(* LS Electric XG5000 project: Forward_Reverse *)
(* PLC LSPLC *)

PROGRAM NewProgram (* task: Scan Program *)
VAR
    Motor_Forward AT %QX0.0.0 : BOOL;
    Motor_Reverse AT %QX0.0.1 : BOOL;
    Start_Foward AT %IX0.0.0 : BOOL;
    Start_Reverse AT %IX0.0.3 : BOOL;
    Stop AT %IX0.0.2 : BOOL;
END_VAR

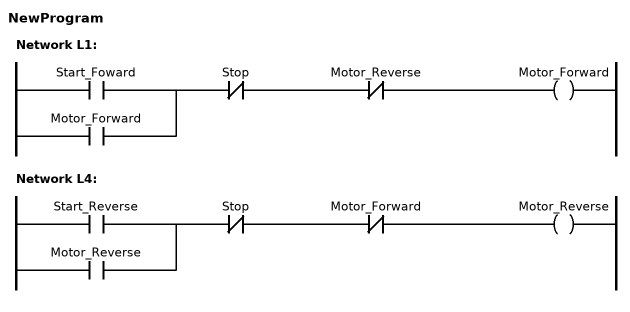
(* Rung L1 *)
Motor_Forward := (Start_Foward OR Motor_Forward) AND NOT Stop AND NOT Motor_Reverse;
(* Rung L4 *)
Motor_Reverse := (Start_Reverse OR Motor_Reverse) AND NOT Stop AND NOT Motor_Forward;
END_PROGRAM